TYPE Stage_t :
(

	 STAGE_INIT,
	 STAGE_ENABLE,
	 STAGE_HOMING,
	 STAGE_WAIT,
	 STAGE_MOVING,
	 STAGE_ERROR,
	 STAGE_RESET
);
END_TYPE

(* stored: Version 1.1.0.1, ProductVersion 3.1.4020.12
   DUT Stage_t: Id {14676720-1ed8-4939-a6d7-49cff4ae6e5c} *)
